FUNCTION_BLOCK NumericValue_IDA (* Input service interface function block for double word input data *)
  (* Description: Copyright (c) 2017 fortiss GmbH, HR Agrartechnik GmbH This program and the accompanying materials are made available under the terms of the Eclipse Public License 2.0 which is available at https://www.eclipse.org/legal/epl-2.0/ SPDX-License-Identifier: EPL-2.0 *)
  (* Version 1.0, 2017-03-20, Monika Wenger, fortiss GmbH, initial API and implementation and/or initial documentation *)
  PACKAGE isobus::UT::io::NumericValue;
  IMPORT isobus::UT::Q::const::IDs::ID_NULL;
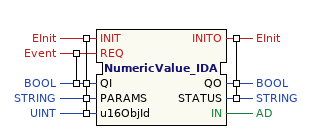
  EVENT_INPUT
    INIT : EInit WITH QI, PARAMS, u16ObjId; (* Service Initialization *)
    REQ WITH QI; (* Service Request *)
  END_EVENT
  EVENT_OUTPUT
    INITO : EInit WITH QO, STATUS; (* Initialization Confirm *)
  END_EVENT
  VAR_INPUT
    QI : BOOL; (* Event Input Qualifier *)
    PARAMS : STRING; (* Service Parameters *)
    u16ObjId : UINT := ID_NULL; (* Object ID *)
  END_VAR
  VAR_OUTPUT
    QO : BOOL; (* Event Output Qualifier *)
    STATUS : STRING; (* Service Status *)
  END_VAR
  PLUGS
    IN : adapter::types::unidirectional::AD; (* Input data from resource *)
  END_PLUGS
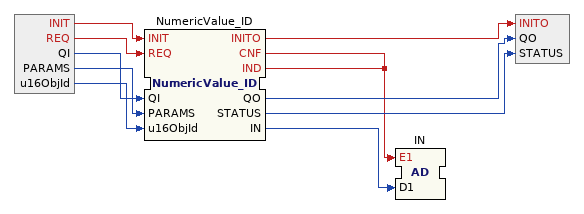
  FBS
    NumericValue_ID : isobus::UT::io::NumericValue::NumericValue_ID;
  END_FBS
  EVENT_CONNECTIONS
    INIT TO NumericValue_ID.INIT;
    REQ TO NumericValue_ID.REQ;
    NumericValue_ID.IND TO IN.E1;
    NumericValue_ID.CNF TO IN.E1;
    NumericValue_ID.INITO TO INITO;
  END_CONNECTIONS
  DATA_CONNECTIONS
    u16ObjId TO NumericValue_ID.u16ObjId;
    PARAMS TO NumericValue_ID.PARAMS;
    QI TO NumericValue_ID.QI;
    NumericValue_ID.IN TO IN.D1;
    NumericValue_ID.STATUS TO STATUS;
    NumericValue_ID.QO TO QO;
  END_CONNECTIONS
END_FUNCTION_BLOCK
